// Mitsubishi GX Works2 project: Pulso_28.09   PLC: Q03UDV

PROGRAM MAIN
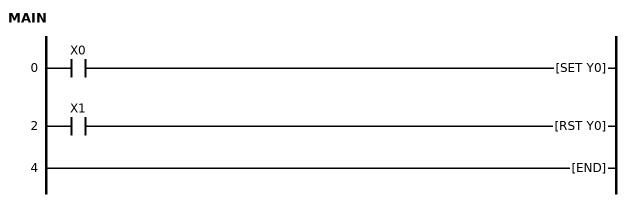
0     LD      X0
      SET     Y0
2     LD      X1
      RST     Y0
4     END
END_PROGRAM
